PROGRAM PRG_FastenerControl
VAR
END_VAR

(* ---------------------------------------------------------
   程序骨架：侦钉状态、请求和结果管理。
   所属任务：Task_CffMain，调用顺序10。
   唯一Owner：PRG_FastenerControl。
   当前阶段：不绑定传感器，不伪造Fastener OK。
   后续实现：状态机、超时、NOK和报警请求。
   --------------------------------------------------------- *)

END_PROGRAM

(* stored: Version 1.1.0.1
   POU PRG_FastenerControl: Id {A2000000-0000-4000-8000-000000000014} *)
